(* IEC 61131-3 sources: ml2plc/benchmarks/st (part 9) *)

(* ---- LSTM2.st ---- *)
FUNCTION_BLOCK LSTM2_FB

    (* Model Inputs/Outputs *)
VAR_INPUT
    input_data : REAL;
END_VAR

VAR_OUTPUT
    output_data : ARRAY[0..2] OF REAL;
END_VAR

VAR CONSTANT
    weights_0_i : ARRAY[0..31] OF REAL := [1.39262271, 2.07329702, 2.0091362, 1.70178938, 2.3850913, 1.12900257, 1.77114773, 1.79174864, 1.94517601, 1.90923738, 1.87943172, 2.05496025, 2.01677155, 1.98114431, 1.29512143, 1.9032824, 2.06803155, 2.26776886, 2.24906993, 2.35914302, 2.58031249, 0.854317784, 2.0349102, 1.86201072, 1.96425331, 1.27948534, 2.47761846, 1.86080444, 2.06046557, 1.88541865, 1.78743565, 2.44109106];
    recurrent_0_i : ARRAY[0..1023] OF REAL := [-0.134004354, -0.148313314, -0.0194474477, 0.0388797, -0.0824599266, 0.0315496214, -0.173172131, 0.0359949544, -0.200757176, 0.109297805, 0.0659822822, 0.0169876534, 0.254330784, -0.00428949948, 0.129118174, -0.0437734537, -0.0245252717, -0.0815731362, -0.0834033787, -0.077183038, -0.0660836324, 0.0495678931, -0.029196145, 0.03283979, 0.0261739939, 0.0130877821, 0.106014706, -0.057191126, 0.0592699833, 0.0329136439, 0.216046751, -0.0511060841, 0.0071357484, -0.0244121794, 0.0280594658, -0.0301723629, 0.0475499704, 0.0748397335, -0.0587395504, -0.168087989, 0.161314234, -0.0552050099, 0.0945079327, -0.107845977, -0.0959540233, 0.00252881669, 0.139446095, 0.0318621695, -0.111325473, -0.0973692015, 0.0295887217, 0.000735154259, -0.0220976807, 0.0224685688, -0.0352836587, -0.031947881, 0.0713648722, -0.147181049, -0.041276142, 0.163752452, 0.163126245, -0.0694158077, -0.0533319078, -0.0770015121, -0.170238152, -0.178571403, 0.0332847945, -0.0801878721, -0.0456461273, 0.0202053282, -0.0822198018, -0.117651939, -0.0558106229, 0.0733473897, 0.0299465898, 0.0360525213, -0.0536533296, 0.0635128692, -0.0457392968, 0.126843438, -0.0655647293, 0.0488459691, -0.0775968879, -0.170379788, 0.061554566, -0.137451679, -0.115184806, -0.00126610929, 0.0082264822, 0.0221565478, 0.049042806, -0.0857262686, -0.0540655181, -0.090015851, -0.238347262, 0.050842043, -0.170883492, 0.0547744632, 0.042925328, 0.066795744, -0.090761885, 0.0645720959, 0.0878244713, 0.195313513, 0.00631635636, 0.0690589845, 0.131412268, -0.0195933655, -0.00472750515, -0.00867333263, -0.0322425812, -0.0256382748, -0.137210175, -0.00508641265, 0.0411479399, -0.0136672538, -0.188457325, 0.110275678, -0.0535120554, 0.148506701, -0.0941733867, -0.0840847343, -0.203250527, -0.00964725297, -0.0456403047, -0.0917202309, 0.0857251734, -0.142379165, 0.0902288333, -0.0697477087, -0.25946781, 0.200249165, 0.0577523112, 0.0731128231, 0.149998024, -0.0543648489, 0.160912603, -0.040147312, 0.0467842557, -0.00688959006, -0.0149163418, -0.0740291998, -0.0424987338, -0.0501250215, -0.076917544, -0.0832854882, 0.129720092, -0.00917770341, 0.154316008, -0.0984195694, 0.0695591345, 0.0279394947, 0.117725901, 0.0648251921, 0.120997198, 0.00961737428, -0.0130183501, -0.0333279334, 0.049932152, 0.0741841197, -0.0766564682, 0.0841158479, -0.0490418077, -0.00928253029, -0.0196176413, 0.131710216, -0.178811699, -0.0807049945, 0.0945211127, 0.0813005269, 0.0478863083, -0.0749040321, -0.0155161619, 0.0436361209, -0.0399981439, -0.00584720029, 0.219137162, -0.0570646003, 0.0864072666, 0.0547209121, 0.19448778, 0.11035566, -0.0152758295, -0.151405767, 0.0672118068, 0.0867983252, 0.0845759436, 0.0431055985, 0.0178876277, -0.055806689, -0.0743876174, -0.0819625705, -0.0752747655, 0.0704117194, -0.00382922404, -0.0398440622, 0.0417721309, -0.0862388536, 0.0705794618, 0.0484335832, 0.173169613, -0.00238036085, -0.0258361753, 0.148217037, -0.0232884251, 0.0270024538, 0.0563735589, 0.126127064, -0.116592243, -0.054894805, -0.174138799, 0.095002085, 0.0277814362, -0.046509631, 0.00551629113, -0.0126956999, -0.034402471, 0.11015445, 0.0495837145, -0.161556005, -0.0879831612, -0.0552681759, 0.0285979733, 0.163931042, -0.0467763692, 0.101849534, 0.0563726798, -0.0478363261, -0.0134126432, 0.0839114934, -0.185348555, -0.0519256219, 0.0111938342, -0.0469942242, 0.0292907096, -0.0607635677, -0.0199214034, -0.0835910067, 0.0188902467, -0.0856332853, -0.0664014295, -0.150778636, 0.232508123, 0.0984602422, -0.112400122, -0.0707815066, 0.00367648201, 0.0512798317, -0.109921589, 0.207549274, 0.162023827, -0.0390811004, 0.0424390286, -0.0276059639, -0.0962381288, 0.0657916293, 0.122452855, -0.145714879, 0.156922311, 0.174932122, 0.104362868, 0.0848342478, 0.0143698901, 0.0799010321, 0.106308773, -0.235139385, -0.082570672, -0.20124191, -0.0119339572, -0.0909275711, -0.0578141734, -0.10269203, -0.093932122, 0.0914303064, -0.107989773, 0.187612101, -0.01330359, -0.0776220039, 0.0276991762, 0.151062503, -0.0498313829, -0.067400828, -0.00874477439, 0.0098327212, 0.0279471185, -0.134616643, 0.102443077, 0.00515093608, 0.0774946585, -0.0788893849, 0.0691870078, 0.0495144166, 0.0123116644, 0.134680301, 0.0235169455, 0.0158374831, -0.0700131357, -0.0892158076, -0.00706590153, 0.00756208412, -0.0815098733, 0.16224964, -0.0743651763, -0.147885278, -0.0525642671, 0.0721946955, -0.00837692246, -0.077373594, 0.0789944157, 0.0923940986, 0.161076784, 0.0733315349, 0.100722194, 0.0398540571, -0.0822396129, -0.113960207, 0.117588356, 0.0800742581, -0.0111245122, 0.0219515339, -0.0255101845, -0.124131009, -0.240380466, 0.0300145727, -0.2196614, 0.0195070971, -0.0691136047, -0.0881249011, 0.0897721574, -0.125163659, -0.190538183, 0.00175063859, -0.0439649113, 0.119778425, 0.0073960349, -0.0287520792, -0.0209456533, 0.00432721013, 0.195701689, -0.0492347032, -0.0886455923, -0.0122433417, 0.0998576805, 0.0985153913, -0.0163457133, -0.0628783479, -0.195168257, -0.0639438778, 0.164951876, -0.112278, -0.0480273664, 0.0445793085, 0.0903970227, -0.137500077, -0.0213923361, -0.0938236639, 0.0234163329, -0.0859521851, 0.0565886721, -0.1431977, 0.0418196842, -0.0795657262, 0.118214853, 0.00396145741, -0.139788032, 0.133322746, -0.025860507, 0.0901994631, -0.132371172, -0.0476551503, 0.0196201466, 0.0488258637, 0.048791565, 0.0862637311, -0.0668302327, -0.0286542438, 0.0713004172, -0.0974688083, 0.0134516265, 0.10718289, -0.0149930362, 0.0711589083, 0.047025796, 0.035104014, -0.055901099, 0.0565550551, 0.148158491, -0.123526365, -0.228604481, -0.161055535, 0.133236721, 0.180309668, 0.0573264062, 0.024110429, -0.0977662504, -0.0378237776, 0.161678582, -0.0324702784, -0.0193747114, -0.0399733596, -0.0443898179, 0.136378944, -0.0683534667, 0.037007682, 0.204772562, 0.0150840413, 0.00119091454, -0.115353808, -0.0508661531, 0.0945357457, 0.00397635065, -0.0107160192, 0.0445148945, -0.153324053, 0.0779764131, -0.0182528608, -0.134156778, 0.113704324, -0.042016793, 0.0408653244, -0.0345638283, -0.104644932, -0.00025787577, 0.195931494, 0.0634211004, -0.0954237133, 0.000879314728, -0.119162239, 0.0455557369, -0.181164652, -0.0286782533, 0.0838612989, 0.00807927363, -0.149410591, 0.0170738958, 0.00178633351, 0.0720130056, 0.0684362873, 0.104216136, -0.0513023771, 0.011758212, -0.176010668, 0.0966927707, 0.0102190599, -0.0279936772, 0.043596521, -0.0417424887, 0.128085271, -0.0604554452, 0.0849098563, 0.0585800111, -0.242956415, -0.163328066, -0.130404904, -0.121299736, -0.0171396304, -0.0231877025, -0.159575537, 0.0178560223, -0.0958106816, 0.0408961512, 0.144970998, -0.120266221, -0.0517051853, -0.0798958912, 0.0248777233, -0.0202759672, -0.00199979614, -0.149970502, 0.0858172476, -0.0259563103, -0.0816580132, 0.10286995, -0.056762252, 0.100706398, -0.0494532436, -0.0494545288, 0.0237438828, 0.0785808489, 0.103829391, -0.0987794846, 0.00639404636, -0.0520768799, 0.0490948707, 0.0426566862, 0.0361592136, 0.0612452999, 0.0584818758, 0.17560859, 0.0293737985, -0.049783133, -0.107105657, 0.108317658, 0.0812257454, 0.0484825969, 0.111484915, 0.0553024188, 0.00590429641, 0.0106472084, -0.0448202752, 0.0259227678, -0.0365177095, -0.0368360095, 0.0979937613, -0.0990265682, 0.0768370628, -0.00803940371, 0.0511335284, -0.10439276, -0.0556471385, -0.111525387, -0.0822637379, -0.158447728, 0.00631242804, -0.0898952037, -0.0103400107, -0.126665518, -0.12826854, 0.164742142, 0.126374289, -0.0623154193, 0.105801776, -0.0670462921, -0.0859524906, -0.165727615, -0.108836487, -0.0711561739, -0.181308746, 0.0773165002, 0.0591216311, 0.0504512489, 0.00781396218, 0.0489371642, 0.112477235, 0.15160735, -0.012935142, 0.131209746, -0.117033251, 0.0818329602, -0.00354715297, 0.10224212, 0.107696757, 0.00897218473, -0.0807351544, -0.00682571437, 0.0395227484, -0.0326741263, 0.00277444068, 0.074753195, -0.0773364604, 0.100228824, -0.0078582773, 0.0254640095, 0.139588684, -0.136924639, 0.0528058484, 0.0296735466, -0.0419536792, -0.0416563302, 0.0534628034, -0.0191842429, -0.0148097789, 0.0523376055, -0.0542180687, 0.0964108631, -0.120417021, 0.038016621, 0.171443269, 0.100414015, -0.152942792, 0.13210088, 0.0675438419, -0.0117004402, -0.0681549385, 0.140697092, -0.0568291806, -0.0730812475, -0.118596427, -0.0816021189, 0.00568043999, -0.0364705734, -0.0795824528, -0.268455297, -0.00127396476, 0.185255677, 0.0253919102, 0.0383441038, -0.0536498129, 0.0324265659, 0.130935684, -0.0526439697, 0.0885849223, 0.0233933069, 0.111991353, -0.0564337634, 0.0322036669, -0.0236973744, 0.138340235, 0.0345056728, 0.0483544394, -0.0399727114, 0.0238587521, -0.0200702958, -0.0636315271, -0.178390726, 0.093400903, 0.0741568655, 0.0728121176, 0.0038592096, 0.0566493496, 0.191387981, -0.0285235178, -0.0280888584, 0.0401902087, -0.0860493332, -0.0164414719, -0.077161938, 0.00620657578, -0.0703452677, 0.0302030519, -0.038376864, -0.0379175022, -0.129299313, 0.0864133611, 0.112249866, 0.00572548434, 0.14621374, 0.0301852543, 0.149874419, -0.0408704281, 0.162906498, -0.00662965514, 0.0628379807, 0.0268993415, -0.000689674052, 0.134167075, -0.313462943, -0.0514584668, -0.107852802, -0.00314436248, 0.0118370224, 0.0500866398, -0.092870526, 0.141352415, 0.0112507679, -0.00922824256, -0.0692459121, -0.00235652924, -0.0174207557, 0.154500976, 0.081347324, -0.00308398576, -0.00189885148, -0.0499526374, -0.0560274385, -0.0403530262, -0.15555121, 0.0442879125, -0.059743192, 0.00816269685, 0.120614648, -0.00293097575, -0.0731150135, -0.0886584222, 0.0900309607, -0.115198389, 0.191818729, 0.103595406, 0.0381124802, -0.0148502458, 0.0115758171, 0.0609838217, -0.0460009836, -0.0733279809, 0.00619584089, 0.0253677219, -0.0612828694, -0.0889660418, -0.036679469, -0.155304044, -0.0361508727, 0.0593941361, -0.0159850381, -0.107755415, 0.205634415, 0.00516803795, -0.0302425101, -0.071119532, -0.0732871741, -0.00382628315, -0.0291780587, -0.0412666611, 0.0520398542, 0.000519843074, 0.177570358, 0.149022236, 0.10058704, -0.0362605043, 0.127544448, 0.0389988348, -0.0245497897, -0.0136824315, 0.0706591606, -0.0728941038, 0.0614774711, 0.0119364653, -0.133704841, -0.000918392092, -0.134823799, 0.0438350029, -0.00247984286, -0.0626151115, 0.09301278, -0.0666331053, -0.0263147596, 0.0359722786, 0.0305371247, 0.054677207, 0.0119109284, -0.0147482157, 0.00910742208, -0.129100755, 0.033809796, 0.00991856307, 0.00350326137, -0.10226763, -0.0163466893, -0.129900768, -0.135179013, -0.064366892, -0.0374643244, -0.0170351807, -0.0269057527, -0.0223082807, 0.0195573866, -0.154327378, 0.0836651251, 0.101992503, -0.266588628, -0.0957774445, 0.127723008, -0.0702769905, 0.000776129775, -0.0205887109, -0.0611850992, 0.102223888, 0.0193744767, 0.0702703893, -0.0131372688, 0.0499369912, -0.13509807, -0.00585971214, -0.0526572391, -0.0965908021, 0.122484364, 0.0293788202, 0.0450509749, -0.0484344773, -0.0140484432, 0.154743597, -0.0609884039, -0.132091016, 0.0942119583, 0.106592871, -0.12995939, 0.0108766314, -0.0612348542, 0.14751406, -0.112796851, -0.0632852614, 0.10222663, 0.00354706054, -0.033328332, -0.124713257, 0.0113556404, -0.279741585, -0.0857560784, -0.157485113, -0.00395657308, 0.0653496161, 0.0413245782, -0.00413726456, 0.0122570768, 0.166194528, 0.111745253, 0.0223836936, 0.00864755362, 0.0349040143, -0.0376916379, -0.0457340293, 0.0522189811, 0.114521392, -0.0617210828, 0.0331743099, 0.115298331, 0.0447754115, 0.142697737, 0.0433601551, 0.0632954091, 0.0451230034, -0.269107699, 0.000234287232, -0.0699387565, -0.016104091, 0.080592148, 0.0290849321, -0.0106361397, 0.00810046121, -0.174048468, -0.085996531, 0.0171728451, -0.03814153, -0.0919195488, -0.0125079993, 0.00758307241, -0.0626493841, -0.00948416442, 0.113764353, 0.0411069244, 0.111225121, -0.00789413322, -0.0439041629, -0.054905504, -0.135183468, -0.0833396018, -0.0639307648, 0.00211562216, -0.0953369364, -0.163012341, -0.134885401, 0.081080623, -0.112399474, 0.0664561316, 0.0931484252, 0.0478505529, -0.0171904434, -0.0378614031, -0.0456895977, 0.12899968, -0.0597828738, 0.0834410861, 0.0139350276, -0.0282864664, -0.0769604295, -0.181071818, 0.214174002, -0.100946948, -0.0732517987, 0.0612714738, -0.197533071, -0.0227342471, 0.0388891399, -0.100754239, -0.00672170753, -0.0207819417, -0.110634871, 0.022637371, -0.01396285, -0.011750361, 0.00330980448, -0.0859773457, -0.000174265006, 0.129387438, -0.139958769, -0.156467378, -0.0922901556, -0.0325083025, -0.0625371039, -0.0629708767, 0.0614186861, 0.0192336366, -0.0547801182, 0.0301011354, -0.0588637106, 0.0513670668, -0.164495796, -0.00147821754, -0.0780117661, 0.0552018546, 0.109413944, -0.00130969961, -0.00898661651, 0.0132659879, 0.0631986111, 0.0843208879, 0.061540179, 0.0394076332, 0.0400769822, 0.00576977246, -0.0982378572, 0.0421557277, 0.113608956, 0.0188576393, -0.0243477058, 0.0602114797, -0.0545240231, -0.0897894204, 0.101281449, -0.154307395, 0.135896564, 0.0464510098, 0.00640968326, -0.021830542, -0.0177672878, -0.0721066073, -0.309531212, 0.0388812348, 0.145754725, -0.0283625945, 0.0946166068, -0.154452384, -0.0263472404, 0.0116467727, -0.0632445514, -0.0424361527, -0.0449868031, -0.0440483689, 0.162283525, -0.141732365, 0.0662780777, -0.0210850425, -0.0168101434, 0.214176998, 0.15372856, -0.0118867746, -0.062056452, -0.000693539158, 0.104848668, 0.120308466, 0.0414873511, -0.112575084, -0.0714760497, -0.0417096615, 0.222792968, -0.110523865, 0.0548756756, -0.117230386, 0.0457057953, 0.0473512486, -0.0799265727, 0.105714075, 0.0468949117, -0.132061332, -0.0291638914, 0.102133185, 0.0477667376, 0.0171793289, -0.0337885171, 0.151557818, -0.0374314077, 0.0159622598, 0.194910049, -0.0489041544, -0.133889884, -0.11275547, -0.173466712, -0.0138423145, 0.13869071, 0.0596037172, 0.062202137, -0.0821835101, 0.0251389612, 0.0879076049, -0.0829390064, 0.0959333256, -0.0619588941, -0.141935766, 0.114354968, 0.155747041, 0.00375959137, -0.0630423576, 0.0245623328, -0.0128721073, -0.103164501, -0.000736813992, 0.0574771278, 0.083872661, 0.0506197587, -0.0941908583, -0.0433398113, -0.00233667111, -0.0455719605, 0.0782523602, 0.173237547, 0.0224949233, -0.0517513119, -0.0378127173, -0.0389218852, -0.0414382815, -0.166335255, -0.110787965, -0.0431358181, 0.0556307398, -0.0059117917, 0.00672180811, -0.00877491664, 0.0884027109, 0.0815280005, 0.0644761026, -0.0395023786, 0.145024762, -0.152458549, 0.0229760204, -0.0113443667, 0.178633645, 0.0435204618, -0.119631179, -0.155641362, 0.169697255, -0.0196635164, -0.0875597149, 0.0888158455, -0.0858875215, 0.112062834, -0.0394157432, -0.120597802, -0.0225557201, 0.0881219059, 0.0495140031, 0.0828080699, 0.00243129907, 0.0277386475, -0.00106827542, 0.0104990676];
    bias_0_i : ARRAY[0..31] OF REAL := [2.26711226, 2.27420187, 2.30581617, 2.31258035, 2.41937995, 2.14668489, 2.35069036, 2.0788188, 1.95626056, 1.9590205, 2.35707855, 2.41049099, 1.97553778, 2.61581278, 2.24078465, 2.34379292, 2.58412099, 2.61249423, 2.82780743, 2.28536749, 2.70651102, 2.23035336, 2.46460962, 2.46926284, 2.27272534, 2.30647492, 2.72902465, 2.39153671, 2.38868213, 2.66885066, 2.01619935, 2.59971189];
    weights_0_f : ARRAY[0..31] OF REAL := [-0.103510261, 0.155920088, 0.000336945057, 0.0438489616, 0.0438292921, 0.0684255958, -0.0156891793, -0.0915879682, -0.150318235, -0.0157852769, 0.165699959, -0.0541729182, -0.130850449, -0.102231637, -0.09064731, 0.185210466, 0.0596044362, 0.0255541503, -0.132748216, 0.168993115, 0.0778170228, -0.178415745, -0.0980168432, -0.111201935, 0.00410218537, 0.0909076929, -0.19583635, 0.177583277, -0.195816249, 0.05490008, 0.129835844, 0.0483838022];
    recurrent_0_f : ARRAY[0..1023] OF REAL := [-0.00691014668, 0.0539467856, 0.0330422595, -0.0597359128, 0.0169141795, -0.0331418402, 0.0173334759, -0.115839541, 0.0169229154, 0.00140885415, 0.0407177694, -0.0358268954, -0.109294459, -0.144246504, -0.000686382409, -0.112673983, 0.204203159, 0.151690304, -0.0307787433, -0.0266794655, 0.118159838, 0.0687537044, -0.196012646, 0.125656754, -0.0728332177, -0.110024385, -0.0255501121, 0.0337689295, 0.12247669, -0.00833526812, 0.0699421838, 0.10112042, -0.0160470735, -0.251208723, 0.0141219553, -0.104823828, 0.0795288607, 0.146455094, 0.193343654, 0.0469122157, 0.00523563568, -0.0152252698, 0.107677527, 0.0577447973, 0.203866184, 0.0566105619, -0.0699815378, 0.0103690829, -0.025823988, 0.0698903576, 0.0937844068, -0.0525806397, -0.0100893909, -0.00210557133, -0.027120579, -0.125489399, -0.0150436275, -0.137994111, -0.0517354123, -0.00446202187, 0.0964010805, 0.0635783747, -0.179122448, -0.0195943583, -0.0458602905, -0.117201932, -0.104822852, -0.0428061485, 0.102384202, -0.0332811326, -0.0195743572, 0.139496908, -0.227235973, -0.0425146483, -0.0722654611, -0.00887431018, -0.132653967, 0.0553128608, 0.112583086, 0.165537104, 0.0365887061, -0.101447128, -0.0985822976, 0.134091511, 0.126952991, -0.0307374429, 0.156312183, 0.0430723652, -0.0509468019, -0.0238420386, 0.0764375478, -0.156924069, 0.207784161, -0.0545833334, 0.0418132134, -0.0283788238, -0.0884652212, 0.0490699746, -0.0942642987, 0.0732667968, -0.030637661, 0.070327282, -0.0578977019, -0.00136273983, -0.0913911015, -0.0634720176, -0.00320455851, 0.0674236417, 0.153130755, 0.0737068728, -0.058094427, -0.0211398825, 0.047294125, -0.0165242814, 0.0421787389, -0.194994301, -0.00844584592, 0.224502295, 0.0124900211, -0.0566204153, 0.14547962, 0.0214617066, -0.0670055449, 0.0452741906, -0.0959712192, -0.20302707, -0.12255279, -0.121577464, -0.243490487, 0.111299828, -0.0271219537, -0.138370499, -0.00303730182, 0.0865178406, 0.036418654, 0.0138794044, 0.168218017, -0.0838619396, -0.0444532298, 0.0891045108, 0.00708426163, 0.0661141723, -0.0399264023, -0.196934208, -0.00761342235, 0.0918690488, -0.0572661683, -0.19526419, 0.0615054481, 0.0232604593, 0.0763470009, 0.00757205719, -0.170795515, -0.0579727553, -0.176360965, -0.0789391994, -0.100149475, -0.065748468, 0.155853912, 0.212572694, 0.0898325294, 0.0844217762, 0.0629207939, -0.0372571982, -0.0432355106, -0.181974009, -0.0866544694, 0.0077539701, 0.0990353674, 0.0708501711, -0.0190058965, 0.0995751917, 0.0896994844, -0.00912527274, -0.0338458568, -0.0137675917, 0.0123393871, -0.0475793704, 0.00175741455, -0.0418805219, 0.115797728, 0.102187678, -0.119467586, -0.0719964802, 0.0550041869, 0.0517715327, -0.0794643909, -0.0289103501, 0.162206873, 0.0127481343, -0.158131227, 0.0304524321, -0.0849102885, 0.0366410948, 0.00384486257, 0.00391263934, 0.0273174196, 0.0815227702, 0.121064574, -0.0600702949, 0.0945892483, 0.057374645, 0.0601622164, -0.0795332193, -0.117707953, 0.0210899487, -0.0372100323, 0.0654684305, 0.0984267443, -0.105141684, 0.138595685, -0.242979154, 0.0243996978, -0.146832377, -0.0938290209, 0.0239801873, 0.124723487, 0.0749439299, 0.0199104045, -0.0626129135, 0.0605645701, -0.112765379, 0.183117643, 0.0728753209, -0.0168619975, -0.0250719804, 0.055014126, -0.0111222807, -0.0467175767, -0.120118842, -0.0719998553, 0.0297824219, 0.0637432635, 0.0930763558, 0.13979651, -0.0786714107, -0.0663307607, 0.0274352431, -0.0654640198, 0.0392157845, -0.0611319244, 0.0636766329, 0.0744584575, 0.0101938117, 0.0555800907, 0.0684161484, -0.0313910916, -0.0375169925, -0.0980222523, -0.138520613, 0.0849486813, -0.1236277, 0.229274869, -0.106394686, -0.104073107, 0.14711982, -0.108186357, -0.0884629786, 0.00385326333, -0.0557541102, 0.0872948691, 0.107587278, 0.0581731871, 0.0215235408, -0.0997304693, -0.0756542683, 0.111098066, 0.0226193108, -0.116672814, 0.0418509804, 0.115937918, -0.0735490248, -0.110052764, 0.063148357, 0.00697960611, 0.0338207707, 0.217933804, 0.059628129, -0.00196746015, 0.123881862, 0.117818907, -0.0192651134, -0.0493695848, -0.0318081304, -0.0192032102, 0.0678166598, -0.00145450607, -0.0869160444, 0.164906725, 0.0981748998, -0.0928812325, -0.0604305677, 0.104643285, -0.142461985, 0.0815763474, -0.00508458167, -0.115501776, 0.0773961246, 0.269783676, -0.172341615, 0.153024822, 0.0490144491, -0.0540101454, -0.0356579125, -0.0566640384, -0.0655708835, -0.0586362667, -0.188088432, -0.0623720735, 0.0904100835, 0.0650910586, -0.0290365405, -0.05520254, 0.0847302079, -0.0487206914, -0.0588986054, 0.0449058786, -0.0469482914, 0.00918797776, 0.0142356111, 0.0266836565, -0.138558552, -0.0684637055, -0.106428206, 0.0228035878, 0.00893711299, 0.00322866905, 0.0695354939, 0.0546293296, -0.0871017501, -0.0162100531, 0.0719157681, 0.0608419478, 0.0179101136, -0.111390203, -0.0720891654, -0.0755965486, 0.0167733729, 0.0292966813, -0.123163752, 0.00929058343, -0.235721245, -0.0745700151, 0.0623340309, -0.0371385068, -0.0765249506, 0.0989028439, -0.139854208, -0.0925003365, -0.0397025943, -0.115456559, -0.116422005, 0.032429643, 0.0281777196, -0.0239272695, -0.0328503177, -0.144181833, 0.0372066684, -0.0524021909, -0.0436877087, -0.144946769, 0.0973152816, -0.107339486, 0.100682661, 0.0554906614, 0.0365729779, -0.0905715972, 0.098124668, -0.0407010354, 0.231915027, -0.103092752, 0.0268508829, -0.00293016527, 0.082363911, 0.0652320087, -0.0384592302, 0.12898241, 0.0402026586, 0.0469526425, -0.0367732197, -0.0941489637, -0.21039243, -0.0243418086, 0.0567742139, -0.0757714957, -0.224011689, 0.111577362, -0.0840680152, 0.00466096681, -0.0797860324, 0.0477439202, 0.0298575554, 0.0669026896, -0.0090283975, 0.112681448, -0.0502874851, -0.00540959276, -0.0274625272, 0.0441634879, -0.0369217657, -0.0101684844, 0.0535784513, -0.00723357126, -0.00442850217, 0.0174251013, 0.0924004242, -0.0299789757, -0.152222574, -0.142336786, -0.0262773167, -0.0686421767, 0.167089716, -0.0872355402, -0.0557465181, -0.113622896, 0.14195551, -0.0551547408, -0.0710106269, -0.067609705, 0.0912378356, 0.0599844456, -0.0631347969, -0.0533212051, 0.0721441358, 0.145896912, -0.0850262195, -0.0618097708, 0.029887341, 0.0855583772, -0.000903251348, 0.0312168524, -0.144762039, -0.0528443567, -0.0244600698, -0.138042107, -0.059540391, 0.0647165254, 0.116018802, -0.158837333, 0.0567534491, 0.0310964324, 0.0519501194, 0.166376859, 0.000156691065, 0.0405331813, -0.0376353115, 0.0910912305, 0.0336197764, 0.0320295431, -0.0283036716, -0.00967699476, -0.0228656419, -0.0633295774, -0.0474807657, -0.0476354286, -0.0262157004, -0.00842537172, -0.0226355828, -0.036474023, -0.144134447, -0.0138616599, 0.0502098948, -0.141214415, 0.0914947763, -0.211922467, 0.108886033, 0.0302329641, -0.0443936884, -0.024401769, 0.178851143, -0.0395925194, 0.109363601, 0.017790867, -0.0280343331, -0.00382982777, 0.00198424468, 0.0132888649, 0.0585306659, 0.0230387188, 0.0412786007, 0.0889222324, -0.122444734, -0.0592958406, 0.061345689, -0.0724695697, -0.17240414, -0.0215452053, -0.11073748, -0.161671206, 0.0069130389, -0.0864949152, -0.0884157494, -0.107923985, -0.149227038, 0.103861548, -0.0224465597, 0.024422098, 0.0677691996, -0.145919502, -0.0570074134, 0.0319532827, 0.0987191796, 0.0601408072, 0.0278520733, -0.146264344, -0.0350774638, 0.0202368796, -0.0724366754, -0.0483524352, -0.156716764, -0.0751653537, 0.0405076034, 0.106280632, -0.090791665, -0.0230285358, -0.0929582193, -0.111961611, 0.016109759, -0.0204031523, 0.0609163716, 0.136724174, 0.0567737892, 0.00902334042, 0.16077508, -0.124572918, 0.0124027627, -0.103831545, -0.0465113223, -0.057945013, -0.117938057, 0.0314415023, 0.0152452486, -0.0766829997, 0.0884116963, 0.0839675665, 0.0765219554, 0.0703505203, 0.0279270336, -0.0127789946, -0.0291803852, 0.0105592217, 0.0371113271, 0.0967723876, 0.0892940015, 0.103656046, -0.260149986, -0.0384903848, -0.0810357556, 0.0938086882, -0.0499689803, -0.0526683852, 0.0961615741, -0.00260981917, 0.00965978112, 0.0354677886, -0.0273469277, -0.0378791988, -0.0684229508, -0.153382406, 0.0829801634, 0.0420659184, -0.0491692908, 0.0548881516, 0.0939008445, 0.0785935223, 0.072916232, -0.0753023624, 0.101734571, -0.212460309, 0.216674268, -0.0828238726, 0.179046914, -0.0126461163, -0.0996344835, 0.0554261804, 0.0543882214, 0.0894713178, 0.0131856054, 0.18864961, 0.0088903252, 0.133240402, 0.0488812737, -0.0503490269, 0.120177239, -0.12674436, 0.0911346078, -0.204793841, -0.0583979376, 0.0430473685, 0.0117439311, -0.100650795, 0.0597399846, -0.183556691, 0.0328893699, 0.0997276679, -0.162350491, -0.0379387476, -0.0467698462, 0.057570409, -0.0352495015, -0.0132564018, 0.0427324548, 0.0986689329, 0.0538132042, 0.000333502423, 0.0106591079, -0.106351398, 0.0680583045, 0.093219772, 0.028425552, -0.0404609889, -0.20924823, -0.127012178, 0.0357946232, -0.0195649005, 0.0538770743, 0.0498228967, -0.056039989, 0.0299009793, 0.0457624719, 0.0841314942, 0.00167563639, -0.0151560055, -0.0918175727, -0.0157458112, -0.252087355, -0.0610392466, 0.118945099, -0.0761914626, -0.059865877, 0.0874174461, 0.145287514, 0.0177363213, -0.207373992, -0.158034712, 0.0130132614, -0.0213055164, -0.110472739, -0.0698485523, -0.00191319175, 0.026409829, -0.149118632, 0.0352956653, -0.0690959916, 0.0712720454, 0.0497274585, -0.0684742928, -0.0192867741, 0.0131304041, 0.0943724513, -0.158797354, 0.0100931283, 0.0212941729, -0.173423976, -0.0672471523, 0.0538061112, 0.125850394, -0.0581939593, -0.0356761925, 0.101517476, 0.0305221472, 0.072131291, -0.051977843, 0.0737764239, 0.0950229913, -0.0675911531, -0.098661676, -0.134873658, 0.0323955193, 0.093537353, -0.0435548872, 0.0345223173, 0.0441020727, 0.0258881748, -0.0267370548, 0.0141971605, 0.0358532406, -0.124594763, 0.0248470921, -0.0100919018, 0.0500047579, -0.0708093271, 0.128508076, -0.0366209187, 0.106708124, -0.00206466648, 0.0805527717, -0.122561544, -0.0874712169, -0.0383777618, -0.0786395073, -0.0780212358, 0.0687881485, -0.0462901331, -0.0869080275, -0.0328290574, 0.114670701, 0.1203302, -0.0302833952, -0.0977141485, 0.0308538172, -0.054454051, -0.0955775306, -0.0812499896, -0.0532917529, -0.047714889, 0.0148271862, 0.0594015457, -0.0969915688, -0.0696531162, 0.0647605136, 0.0158956926, 0.00915151369, 0.16740869, 0.111624435, -0.0313705765, -0.126204967, 0.166225314, -0.00429002754, 0.00159279886, 0.170427188, -0.0651404411, 0.0322218463, -0.107634276, 0.110197365, 0.0253799651, 0.0844260231, 0.109976798, -0.0586437285, 0.0578876138, 0.000859050546, 0.189837858, -0.0570421889, -0.170068368, -0.0814624578, -0.0846147761, 0.0692067817, 0.0624997802, -0.227033526, -0.0656075999, -0.0454960801, -0.0364593938, -0.0984016657, 0.139481351, -0.0299721137, 0.0211200267, 0.0929757655, -0.162706748, -0.192191154, 0.194119602, 0.146404952, 0.0726765618, -0.0705825686, 0.000404240564, 0.00767246261, 0.0835697502, -0.0302281529, -0.0174284484, 0.0485032201, -0.120143197, -0.108964629, 0.0507510044, 0.00870033167, 0.0645659417, 0.108325213, -0.0504615642, -0.0399887264, 0.0522538908, 0.103842363, -0.0575898327, -0.0733171329, 0.0778556466, -0.0311737508, 0.000791670987, 0.053147953, 0.000775715336, -0.0727582201, 0.059283942, 0.015961254, 0.0980835333, 0.153303385, 0.0523465499, 0.200393319, -0.0961034298, 0.00924751814, -0.102561079, -0.127784446, 0.0216288883, -0.0499887094, 0.0408567637, 0.0934649706, -0.0518678166, 0.132874012, 0.0137811955, -0.05145818, 0.0129512828, -0.139415756, -0.143087536, 0.068125844, 0.10787306, -0.057314042, -0.0380743705, -0.0627397448, 0.130972728, -0.0196755826, 0.0785539597, 0.122383311, 0.0626117215, -0.0613358766, 0.0130844237, -0.0416473523, 0.0771606714, -0.053707961, 0.0782196, -0.00344187161, 0.102742925, 0.0139414081, -0.155407608, -0.0412477255, 0.0853889138, 0.063173607, 0.116590202, -0.110537179, 0.00120887649, 0.112075336, -0.0691253319, -0.0917270258, 0.0188949592, 0.00672117434, 0.0868049711, -0.121678926, 0.116180249, -0.0147003271, -0.0895797387, -0.135892138, -0.141551331, -0.212871507, -0.0520402603, 0.0142919831, -0.088278383, 0.0244035851, 0.0466132648, -0.0750784948, 0.106897034, 0.106365465, -0.0986929387, 0.168738917, 0.0507040955, 0.00279272767, 0.0927622467, 0.226838261, 0.0705733225, -0.152726993, -0.0682013631, -0.069567509, -0.106382623, -0.0238234401, 0.0889748037, -0.095707342, 0.0320834182, 0.0533372127, 0.0397444218, 0.173014328, 0.114501618, 0.050176464, 0.0578774475, 0.0132526672, 0.100262016, 0.113684908, -0.127054498, 0.016781047, 0.105807446, 0.160546854, -0.0204436425, 0.0449761264, -0.00650018919, -0.0162856318, -0.031046655, -0.00719706295, 0.17228359, 0.0929863527, 0.112568557, -0.0106027573, -0.0801606029, -0.00430984143, 0.0905482695, 0.102497414, 0.022951575, -0.0023685242, 0.101059511, -0.123741455, -0.0253990814, 0.00617785938, 0.224820018, 0.0564163029, 0.0227698721, 0.0183891784, -0.193179756, -0.048081845, -0.00418907218, -0.0182756223, 0.0594953559, 0.116223007, 0.083689943, 0.0758306682, 0.0600401387, 0.0057036127, -0.119169444, -0.00241687289, 0.049240943, 0.0222266763, 0.0222300421, 0.0184250548, 0.137113541, 0.133112341, -0.0405313745, 0.0703310296, -0.0368162692, -0.00698137842, -0.0782028064, 0.154308647, -0.0416583829, 0.0667509288, -0.0523070544, 0.000271657365, -0.148217291, -0.011399786, 0.0411178507, 0.0403273664, 0.182938606, 0.00969816186, -0.0497058183, -0.0412162356, -0.0586917587, 0.136667043, 0.0978190973, -0.0634948984, 0.0585792921, -0.0983795375, -0.0980659947, 0.0711884275, 0.0689789802, -0.109272763, 0.0259555485, 0.0922681913, 0.0452702269, 0.0214219354, 0.0569992065, 0.0292213559, -0.0258827768, -0.0412379466, 0.147309318, 0.0441662334, -0.0152443759, 0.00304972567, 0.182876348, 0.164139763, -0.111702725, -0.0858073086, 0.0243306477, -0.0263965055, -0.08150056, 0.0267791264, -0.0301363561, -0.110263094, 0.0477498025, 0.0285967328, 0.0422384776, 0.145023987, -0.0232882276, -0.109742552, 0.0407254286, -0.101167023, 0.087719284, -0.144451484, 0.0783894286, 0.116550274, -0.0671435595, -0.0849284753, -0.00986922067, 0.0360355005, 0.161055446, -0.118753619, -0.0674274117, 0.0250015743, -0.0504739732, 0.136040404, -0.160468519, 0.0275609754, -0.0788998529, -0.0405119434, -0.00997654907, -0.061767187, -0.053517133, -0.0994137824, -0.0556045212, -0.0925223976, 0.161830351, 0.0968106836, 0.0508179069, -0.0246349927, -0.0123783387, 0.0485562719, -0.0574627705, 0.0263824128, -0.120863646, -0.0710439906, 0.0614336506, -0.106016003, -0.0335879326, -0.0433921926, 0.0639650673, 0.0271945707, 0.0527300388, 0.0320915915, 0.013170423, -0.08443138, 0.248558924, -0.0503826216, 0.106785677, -0.046431087, 0.103803217, 0.0041458183, -0.0421562381];
    bias_0_f : ARRAY[0..31] OF REAL := [1, 1, 1, 1, 1, 1, 1, 1, 1, 1, 1, 1, 1, 1, 1, 1, 1, 1, 1, 1, 1, 1, 1, 1, 1, 1, 1, 1, 1, 1, 1, 1];
    weights_0_g : ARRAY[0..31] OF REAL := [1.47532678, -1.70458651, -1.47144258, -1.44691277, -1.68858755, -1.54678094, 1.4575063, 1.77509093, 1.5990113, 1.71160305, -1.5320437, -1.79037261, -1.77602446, 1.70425713, 1.4617672, 1.54794741, -1.52839839, 1.55297565, -1.90853524, 1.71287596, -2.10243273, 1.36646223, 1.82073891, 1.9412576, -1.69837666, -1.66724396, -1.99537337, 1.69469917, -1.80649602, -1.47025287, 1.49180543, -1.93371117];
    recurrent_0_g : ARRAY[0..1023] OF REAL := [-0.101195998, 0.08740969, -0.104587115, -0.16821076, 0.174443915, -0.035774447, -0.0947507322, 0.0378404111, 0.0557015277, -0.0394512936, -0.207284242, -0.197577581, -0.0711208954, -0.120538749, 0.0129681649, -0.0769899487, -0.0140917841, 0.00214586221, 0.00265539065, -0.123874903, -0.107705243, -0.105937153, -0.0518222116, -0.0369259045, 0.0763554201, -0.0299211461, -0.0788105503, 0.117140636, 0.00431261165, 0.0359783769, 0.00918749906, -0.104668915, 0.061548844, -0.0556093194, -0.0334143862, 0.0841006264, -0.0666153282, -0.0459342971, -0.0507918485, 0.0554375648, 0.0217144638, 0.0350073129, 0.124298088, 0.0216758177, 0.120086238, 0.0596877821, -0.0242632702, 0.0876686648, 0.0902777761, 0.0481038094, 0.204886943, 0.180912375, 0.0283590574, -0.00545403361, -0.111476384, -0.0184426904, 0.0296593215, -0.0534377694, -0.0470365658, -0.0600505061, 0.0377211198, -0.0949909091, 0.160191432, -0.0323576629, -0.00774259027, -0.000638007885, -0.0570991226, -0.00242817705, 0.0460335501, -0.0124942036, 0.255657285, 0.0184760075, 0.083474122, -0.138274193, 0.0288563892, 0.0561495312, 0.10814105, -0.0252166167, -0.083617121, 0.00315840216, 0.134269193, 0.080687955, 0.0888233185, 0.0208418351, 0.0151973907, -0.0696730837, 0.254600137, -0.126226783, 0.00475102197, 0.0205613524, 0.0766184479, 0.0583407693, -0.0356217064, 0.0329036042, 0.00880802702, 0.0259327479, 0.0302957594, -0.0485900454, -0.0475254133, 0.0427846983, 0.14055638, -0.125194758, -0.230593339, 0.115369402, -0.009178821, 0.0961865857, 0.0861247405, -0.0569514222, -0.0642841905, 0.0787181482, -0.000574963633, 0.00898596738, 0.0703639537, 0.0666252524, -0.082310304, 0.0077218432, 0.0239734557, -0.154473484, -0.130902037, -0.138917118, 0.168707773, 0.0168054793, -0.241201326, 0.0562871881, -0.0551889241, 0.0774001628, 0.0454477295, 0.0527046323, 0.192182556, 0.0634233505, 0.0726593807, -0.0730486736, -0.046287708, 0.0937241539, 0.155822381, -0.0986693949, 0.10592638, 0.0549062192, 0.0108801452, -0.0758548081, -0.150141403, 0.000112835725, 0.168501094, 0.0566198267, -0.000829054043, 0.081648834, 0.0720061287, 0.00562748406, -0.0315910913, 0.0916485265, -0.0881970823, -0.0454844274, 0.115997486, -0.0706517994, 0.200185716, -0.212817028, -0.266671538, 0.0280515496, -0.0507685766, -0.0832299516, -0.0272886436, -0.0584619641, 0.0404174477, 0.139308289, 0.104658842, -0.083959721, 0.0130339842, 0.0628424138, -0.0578840524, -0.0111292899, -0.0674168542, -0.0567888021, -0.0487619378, 0.0660481378, 0.140314907, -0.103330687, -0.077637881, 0.0232625715, 0.16300194, -0.0148641821, -0.121850781, -0.0120066088, -0.120630994, 0.0325469822, 0.00378151797, 0.0231334269, 0.0288972799, 0.117997028, -0.00443882123, -0.154459015, 0.0336177275, 0.0930437893, -0.00218074629, 0.131201416, 0.095992431, 0.115522057, -0.0244959947, -0.00682251481, 0.0696546957, -0.0206905808, -0.0148855159, -0.0281523354, -0.03817432, 0.0418252461, 0.0572236478, -0.0574149303, -0.109414637, 0.0453919359, -0.000927357178, 0.0428337641, 0.0247878674, 0.0959960148, -0.00927572511, -0.0164810531, -0.116284199, -0.0459703058, -0.0627707541, 0.0265134163, 0.0581545085, -0.00378958462, 0.0373996682, 0.0825420693, -0.0857948065, 0.0619786419, 0.081787698, 0.108454175, 0.0945709571, -0.051475592, 0.0921381786, 0.170338392, 0.137564644, -0.132172644, 0.0645276457, 0.154890299, -0.0760021806, 0.096898526, 0.0867238268, 0.109539069, -0.0057261046, 0.060632281, -0.100636743, 0.157683015, 0.0451725535, -0.00428324332, -0.0746827871, 0.0471339598, -0.0752350464, 0.069367975, 0.047093872, 0.00814475119, 0.011384381, 0.0659590662, 0.156899557, -0.0580012202, 0.085925512, -0.0214249622, 0.0120120468, 0.113536887, 0.0602683052, -0.0160956811, -0.0338802151, 0.0308419038, -0.0770991966, 0.000288646523, 0.0453838557, 0.0851812661, 0.0191567522, 0.0233700275, -0.121437192, -0.0659240335, -0.123420395, -0.0978944823, -0.0577415749, -0.0328979529, -0.0636603981, -0.00405571982, -0.0314529873, -0.020198442, -0.0146561153, -0.0762880072, -0.0999139771, 0.0514613762, 0.0256823711, -0.0942612588, -0.052791819, -0.133564845, 0.0861075073, 0.00868083257, -0.00935054384, 0.0302694831, -0.0317124836, 0.087807633, -0.0803157836, 0.089592196, -0.0941260234, 0.0717165917, 0.0632364899, -0.214625821, 0.137252107, 0.209107444, -0.117832825, -0.00798236765, 0.0595166907, 0.118651874, -0.108172223, 0.136428297, -0.18883127, -0.107870199, -0.0385832936, -0.206498623, 0.0613527596, -0.00105835567, 0.136841521, -0.0176947806, 0.00627136417, 0.0683735684, 0.0605167933, 0.0425770134, -0.00393029675, 0.00458816718, -0.0597686134, 0.0324797593, -0.0304794982, -0.0699171275, -0.0795711279, -0.0220978875, 0.11555858, -0.0186585672, 0.0740450099, 0.0289000161, -0.0231691636, 0.125412941, -0.0254150778, -0.0975785479, 0.0826669931, 0.0427691564, -0.0265431367, 0.0233916827, 0.0275735483, -0.159331188, -0.0835884213, 0.0867214575, 0.0581048802, 0.0400546007, -0.11298833, -0.0843894854, 0.0884476602, 0.156565502, 0.0398587845, 0.084373489, -0.167539656, 0.0533768237, 0.180099636, -0.0643721148, -0.022131959, 0.0352704972, 0.102284059, -0.129944429, 0.0652202368, 0.0329418108, 0.0671919212, 0.0213613939, -0.041750174, 0.140751526, -0.010692168, 0.108571574, -0.0590898506, -0.00340850884, -0.101751246, 0.0585011132, -0.0625699461, 0.0747210979, 0.143278256, 0.0285833869, 0.000918021193, 0.0832627043, 0.0124035478, 0.00828075409, -0.0645460263, -0.0208687484, -0.0479471907, -0.0879585519, 0.00869457796, -0.0489250496, 0.0110164564, 0.0660134107, -0.0409986079, -0.0835550651, 0.108670741, -0.0402804874, 0.0745845065, 0.0347721204, -0.0930110365, -0.0466776416, 0.0181542635, -0.122449115, 0.0457023606, 0.0551486239, 0.0993403047, 0.0452728644, -0.0912225768, 0.177634746, -0.0193397272, 0.0517804064, -0.078884609, 0.0770803168, -0.026274981, 0.115404844, -0.0222992562, -0.0548713244, 0.115336612, 0.102776915, -0.105107367, 0.0272116847, 0.0181901883, 0.116371438, 0.0772981793, -0.0657144263, 0.0702497438, -0.0933898166, 0.00560039189, -0.117238283, 0.043919649, -0.0706500262, -0.036055591, -0.103364304, 0.0620049611, 0.122532926, -0.0542505234, -0.0309813488, 0.112967849, 0.00626176875, -0.0412489027, 0.000259818044, 0.1122576, -0.022883717, 0.0698174983, 0.0954817906, -0.0475088432, 0.0141142579, -0.0512579754, -0.0754119679, -0.0424957797, 0.0419287719, -0.054218974, -0.156465426, 0.114787057, -0.0610668324, 0.0348946378, -0.040694993, 0.121415451, 0.0283232052, -0.0169020146, 0.139543638, -0.170662105, -0.119277015, 0.0594007708, -0.0582244582, -0.0817419291, -0.0981166661, 0.00173791777, 0.00693563698, -0.0207109731, -0.035633482, 0.0308553185, -0.0928787142, -0.0212399177, 0.0114278868, 0.136616603, -0.0549275205, 0.0995251387, -0.0262963269, 0.0154484715, -0.0506038368, 0.015139862, -0.0465807803, 0.0256181471, 0.0665449798, 0.0268637985, 0.136133835, 0.132263571, 0.0828409493, 0.00177018531, 0.188435555, -0.131212503, 0.0970125347, -0.127591342, 0.0796364471, -0.0402331352, 0.0689072907, -0.0653174818, 0.0493306741, -0.139246956, -0.0419746451, -0.0420375466, -0.133270577, -0.0126191825, 0.106959179, -0.0525025129, 0.0485690534, -0.0125091951, 0.0833685473, -0.0323823877, -0.0772480667, -0.0500528924, -0.204458624, 0.0348587632, 0.200497746, -0.0761522502, 0.0727544576, -0.0308812261, 0.0495476648, -0.146705776, 0.0997447371, 0.012238658, -0.00608632155, 0.150759101, -0.123230845, -0.0151646882, 0.0577027462, 0.0434368625, -0.0141762858, -0.200296491, 0.0534211285, -0.011844527, 0.189423949, -0.107985377, 0.0767114758, -0.135413483, -0.00799088273, 0.134802759, -0.0511588715, 0.0691743344, 0.105821721, -0.0770135447, 0.0278117098, 0.00748841185, 0.0431736782, 0.022644151, -0.0930894092, 0.0724659637, 0.119439431, 0.157009006, -0.110694274, 0.0888616964, 0.0203899164, 0.0554994904, -0.0155844046, 0.0935843065, -0.0437429696, 0.0356643498, -0.00294274278, -0.0150379483, -0.152130276, -0.0716923475, -0.221969858, 0.102691673, -0.0195766296, 0.0772279948, 0.0226173997, 0.0137649449, -0.0166043434, 0.116271779, 0.0191773064, 0.00167295639, 0.0734597445, 0.0365498513, 0.0512108281, 0.144751921, -0.0385083035, -0.0588598065, -0.189036906, -0.14177978, 0.0120348353, -0.0084497435, 0.220320597, 0.0226446763, -0.248947561, 0.139383212, -0.0020379154, 0.0696443245, -0.0780093148, -0.0792569518, -0.0160436984, 0.0795049742, 0.0932552516, 0.0753452033, 0.0848368406, -0.00240107533, -0.033641424, -0.0348135754, 0.0561227389, 0.147689387, -0.0594362281, -0.0409766734, -0.250746489, -0.160236001, 0.0386024341, -0.0686084852, -0.0440940112, 0.0674488544, -0.210844234, 0.0464956835, 0.0757730156, -0.0683382824, 0.0804399922, 0.0413802229, 0.0806305632, 0.0221607983, -0.132880241, 0.0989559144, -0.118918777, 0.0531449281, 0.0418806486, -0.0401233248, 0.0478454567, -0.0536536165, -0.00559705123, -0.0308934376, 0.0934929922, -0.0454997756, -0.121145718, -0.0170345623, -0.0106199561, 0.150425464, -0.0529386513, 0.067161046, -0.0163639486, -0.0500465147, 0.103452504, 0.0317030214, 0.0288870297, -0.011946328, 0.0184828602, 0.139818698, 0.101647899, 0.1074147, 0.0303774215, 0.134888709, -0.179935634, 0.036726281, -0.10821747, -0.142873049, -0.0262996051, 0.0476385057, -0.0365874916, 0.111659452, 0.0944161266, -0.0142952949, -0.0806843117, -0.0428597666, -0.0658241659, -0.114456557, -0.106830753, -0.0586995706, 0.0279622488, 0.0323923454, -0.00418315269, -0.131964132, -0.0308927745, -0.0672691539, 0.0376390964, -0.0317809209, -0.147463486, -0.0706574917, 0.0185221247, 0.132252961, -0.158320606, 0.026732469, -0.10199368, -0.0534288362, -0.0309845041, 0.100389093, -0.134254992, 0.00933926925, -0.046615012, -0.12006966, 0.0782608092, 0.0736895055, 0.0822508186, -0.0227471944, 0.0878217146, -0.137264773, -0.1176171, 0.0138121042, 0.0491721779, 0.0136306696, -0.090548791, 0.0630058348, -0.136406288, -0.101197541, 0.0404558256, 0.090086326, -0.128530398, -0.226135164, 0.109265037, -0.0687788427, 0.176857248, 0.0773077458, 0.0409816019, -0.0806122348, -0.0451379567, -0.0299756341, 0.140983731, 0.00555554172, -0.0402856506, -0.084920913, -0.09508463, -0.0965267867, -0.0849358514, -0.0511886589, 0.0146661261, 0.0156131554, -0.0376326963, -0.0671210811, 0.0224287175, 0.137774587, -0.00228940486, 0.0465276316, -0.130178899, -0.149012893, 0.130293623, -0.0280530471, 0.0527597964, 0.21135141, -0.200008243, -0.0908918828, -0.0363020897, 0.0601692759, -0.0125749074, 0.0811389834, 0.17963928, 0.0170890167, 0.207968205, -0.0548401587, 0.0640945509, 0.00915475748, -0.00665144948, 0.0521441624, -0.0598076954, 0.125235885, 0.103107899, -0.0512448139, 0.0199147407, -0.102051727, 0.00533230044, 0.0623953715, -0.0797764882, -0.00129370275, 0.239951834, -0.0897608474, -0.0809930637, 0.0116302716, 0.0264315549, 0.00502448808, -0.0133893285, -0.0398890302, 0.0280222762, 0.0427577049, -0.0401622653, -0.029694058, -0.00408209302, 0.0222895369, 0.0128808133, 0.137052923, 0.00298324437, -0.0114676105, 0.0736051723, -0.140455097, 0.0202825014, -0.02705306, -0.245139763, 0.212917298, 0.104035825, 0.0293759983, -0.0546719022, -0.0314423367, -0.0398630574, -0.0343876965, 0.0905116275, -0.0775412396, -0.129571766, 0.0111265779, -0.127151802, -0.173279762, -0.0682864934, -0.0263398364, 0.0888700038, 0.209845588, 0.051952444, -0.0745497346, -0.185133874, 0.100421809, -0.0359647982, -0.100239962, 0.0507267825, 0.0249746833, -0.0182546433, 0.0273244902, -0.00399943395, -0.024655791, -0.0122731468, 0.200671896, -0.00162600097, 0.0544531643, 0.00520347059, 0.0765429288, -0.167934522, 0.111238033, 0.0929705277, -0.00967021845, -0.0453585982, -0.102070257, 0.112714708, 0.0161449425, -0.129575238, -0.0770349205, 0.0931738392, -0.0932359025, 0.115253128, -0.152637616, 0.0158179048, 0.041739326, 0.103671372, -0.0748060644, 0.0285792667, -0.011899136, -0.0192917511, 0.107791625, -0.0256559402, -0.0543608293, 0.0164244436, -0.0119684432, 0.0224394947, -0.145458579, -0.0641392097, -0.137857869, 0.0793515444, -0.0232694242, 0.0881254748, 0.139484107, 0.0756044835, 0.125058889, -0.00860834494, -0.0920527279, -0.100648604, 0.0184238963, 0.0770169795, 0.0118718268, 0.111209154, -0.113483764, 0.0125254337, -0.0266479366, -0.0571810752, 0.0200069863, 0.124276526, 0.0205191262, 0.0164585561, 0.133350834, -0.00794353709, -0.048325561, 0.0614461824, 0.0337038003, -0.113049902, 0.0363934785, -0.0499502607, 0.0158293881, 0.0611683168, 0.0159349889, -0.124337569, 0.0816555843, -0.0228196569, -0.0540381968, -0.00830301642, 0.0457908213, 0.0331352726, -0.0895112082, 0.00246492564, -0.107790858, -0.0560132973, 0.11573261, -0.0372891389, -0.111539595, -0.0485297851, -0.0968310386, -0.0706709251, 0.0666795596, -0.11741551, 0.0311872456, -0.0177999716, 0.0229795799, 0.0683093667, -0.04996939, 0.0947744995, 0.0472060777, 0.0167367272, 0.0973566622, -0.0538218617, 0.0466017947, -0.0330167077, -0.0814527273, -0.0711240023, -0.0872239992, 0.0632802621, -0.0083680097, -0.0674064085, 0.0238934588, -0.0249120407, -0.0205953475, -0.132834002, -0.155904874, -0.20259355, -0.0278226659, -0.146687314, 0.0802839473, -0.224116221, 0.0802529827, -0.0681261495, -0.0971475542, -0.00637515821, 0.0898840725, -0.0242172033, -0.0200051516, 0.0198571607, 0.0626354143, -0.0625288486, 0.0788489282, 0.0189317074, 0.185568005, 0.000117650256, -0.0706626996, -0.0232296046, 0.0265699401, -0.140608713, -0.0798913389, -0.0144935483, 0.0150925051, -0.0770403296, 0.0461982638, -0.0743894279, 0.0112759992, -0.0415325053, -0.0902260616, 0.0242120959, -0.0101395501, 0.0574476793, 0.0817934275, -0.119240142, 0.00109685957, -0.0366540477, 0.180904225, -0.0508034974, -0.0597405396, -0.00300559308, -0.0296302028, 0.0939078331, 0.0482150204, -0.00707970513, 0.0974167213, -0.0386451483, 0.0357006602, -0.0137596354, 0.202047825, -0.065607585, -0.0113760866, 0.0209448077, -0.0308414511, 0.0818564594, 0.035646081, -0.127649605, 0.105054356, 0.0557748713, 0.00202266965, -0.0665288493, 0.052466169, 0.037145067, 0.0144229438, 0.0539823025, 0.0187405162, 0.0615465529, 0.0469304807, -0.065950945, 0.0401757248, -0.0292687323, 0.158052534, 0.0467117839, -0.064893201, 0.182949245, 0.0275977291, -0.171592563, 0.06078564, -0.0222570412, 0.0590536557, -0.0516086444, 0.0321202911, -0.126681581, 0.0127856554, -0.0842492506, -0.0825054348, 0.145829186, 0.0492514409, -0.021345092, -0.0882940814, 0.219456479, -0.164974764, 0.114569366, 0.084793061, -0.0892998874, -0.0848865286, -0.0151299872, 0.10800042, -0.0836073011, -0.0394540206, -0.00415410474, 0.0545243472, 0.113440655, 0.0142033203, 0.0992297381, 0.0700212419, 0.0218305327, -0.0960413069, 0.0179279074, -0.0658347681, -0.0156512503];
    bias_0_g : ARRAY[0..31] OF REAL := [-0.581836522, 0.309231728, 0.562823296, 0.627700269, 0.377331227, 0.598591506, -0.602125108, -0.303565025, -0.210975483, -0.289409161, 0.45574379, 0.347700447, 0.275302798, -0.5403862, -0.575578272, -0.550802469, 0.286279172, -0.627842605, 0.461831361, -0.275645137, 0.570479512, -0.615097225, -0.421455711, -0.499417245, 0.348250419, 0.679803789, 0.502462208, -0.518211007, 0.372529656, 0.596038401, -0.266079992, 0.497252136];
    weights_0_o : ARRAY[0..31] OF REAL := [1.76166964, 2.15148592, 1.80391347, 1.68124664, 2.52235556, 1.41236889, 1.65919316, 1.83199465, 2.17834687, 1.65460563, 1.72433054, 2.19740796, 1.8024863, 2.31803036, 1.70240915, 1.55125129, 2.21101999, 2.17488194, 2.62146235, 2.56662989, 2.68313241, 0.862560272, 2.02623749, 1.8731904, 1.98365009, 1.40244126, 2.40513897, 1.74895322, 2.16502452, 1.9363879, 1.95291567, 2.40807748];
    recurrent_0_o : ARRAY[0..1023] OF REAL := [0.00940295961, 0.00755411293, 0.115096495, -0.042677924, -0.0687995777, -0.072212413, -0.0272679329, 0.00926187169, -0.0322404131, -0.230642751, 0.10464444, -0.118317537, 0.0643291026, -0.0847248659, -0.110454835, 0.065530844, -0.0409047455, -0.079811722, 0.0585166439, 0.0876166224, -0.0146481553, 0.0276156012, 0.0437087826, 0.0136683295, 0.122135736, -0.0417108536, 0.0472377948, -0.0826558396, -0.0739040002, -0.0169733446, -0.0704516172, -0.111660339, 0.0013261399, 0.032797996, -0.107126579, 0.051768031, 0.168218851, -0.117840573, -0.00133558537, -0.156737015, 0.00473470287, 0.0387410335, -0.0619333275, 0.0416263752, 0.158205613, 0.0598703958, 0.0712381601, -0.0656233057, 0.147444651, 0.0920717269, -0.0842068717, -0.0531333908, 0.0637576878, -0.0327701457, -0.00259020133, -6.20728533e-05, -0.0932620242, -0.136093467, -0.0542191677, -0.0130609386, -0.0714226291, -0.139094964, 0.0650555268, -0.0779461116, 0.0727291405, -0.0236136429, 0.0512026139, -0.101979688, 0.00239524571, 0.0366442576, -0.0302348658, 0.0942990929, -0.0132932235, -0.0642298311, 0.0192060657, 0.0130893327, 0.101625614, 0.200168759, 0.0517889932, -0.108799636, 0.104390532, -0.0586065203, -0.163236856, 0.0647632331, -0.0528851151, -0.107174575, 0.0846626312, 0.037532419, -0.049235642, -0.0950798392, 0.191777244, 0.0884989724, 0.000524577685, -0.0158200487, -0.0106198462, -0.102214061, 0.0069015082, -0.0446161591, -0.0392294414, 0.0153008103, -0.027325429, -0.0261812173, 0.0347592905, -0.0386674777, -0.0300151668, 0.002856954, -0.00180103246, 0.0520746112, -0.00637343619, -0.028616976, 0.0337644443, -0.0843739882, 0.0802535638, -0.0490648001, -0.0998648554, 0.0383425839, -0.0290285107, 0.145915732, 0.00134465739, 0.101120107, 0.182724848, 0.138152152, 0.0405496918, -0.0204477198, 0.0529464185, 0.049938079, 0.0684493631, 0.065276593, -0.00253880629, -0.0155425929, -0.037788067, -0.0378959365, 0.0827185288, -0.164564133, 0.0313715376, 0.0749724954, -0.0116761904, 0.0597785451, 0.0476476401, 0.108241357, -0.0507849157, -0.077297315, -0.00137838325, 0.059471447, 0.0385285877, -0.0541518517, 0.0803878233, 0.0667919442, -0.0593200326, -0.0991778895, 0.0175430924, 0.0742868111, 0.0518188477, 0.00270438683, 0.00619300222, -0.0744272992, 0.04556676, -0.0101611707, -0.0633157417, 0.0911582336, 0.0333724804, 0.0274891406, 0.090359278, -0.0250894763, -0.0330442227, 0.0266552437, 0.119048312, 0.0323781371, -0.0843255669, 0.136369541, -0.0256569721, -0.0414893776, 0.0121494886, -0.00654248102, 0.0232459698, -0.00572938658, -0.0533263944, -0.226630121, -0.157875374, 0.0423009694, -0.0904081017, -0.0658113956, -0.151652411, 0.0201764442, -0.0914419144, -0.221003428, -0.00242811069, -0.0150172506, 0.00472717499, 0.025153067, 0.0449665263, -0.00235806056, 0.079561159, -0.00979024544, -0.032114543, -0.0120351668, -0.0658440515, -0.0523885936, 0.0321432129, -0.0523841158, 0.0984722227, -0.0391403213, -0.144826144, -0.0854723975, 0.00218068436, -0.0135808857, -0.03519921, -0.000386994798, -0.0123389661, -0.0385522321, -0.0213163309, 0.0617649332, 0.0749436319, 0.0909294337, 0.0126738595, -0.0654598102, -0.0385108218, -0.0317040943, -0.109090902, 0.0275919586, -0.0637576133, 0.0479899794, -0.0208571032, 0.0530534722, -0.0127447946, 0.0714634806, 0.0186050329, 0.132866919, 0.047393024, -0.164494514, -0.0709982663, -0.197920769, -0.0988798514, -0.154706299, -0.00919868704, 0.135501906, -0.0794674754, 0.0428844541, -0.0342918821, -0.00617858162, 0.0376018286, -0.0680695921, 0.0221220106, 0.0718257576, 0.118553676, -0.050622128, 0.0384315327, 0.0652998835, -0.204144284, -0.0725613013, -0.0885725841, -0.0328807719, -0.0790686682, 0.0327409133, -0.0627308935, -0.0589160621, 0.107908778, 0.105854571, 0.0165748075, -0.153165773, 0.169386417, 0.0277452115, -0.0437977612, 0.00759721361, -0.0423627906, 0.0660784319, 0.0508499742, 0.143870711, -0.00561960228, -0.023442572, 0.0437386408, 0.00149761862, -0.000399552286, -0.0776806548, -0.0184591748, -0.0243691169, 0.0632502511, 0.0728501529, 0.22410582, -0.0715147927, 0.0263980404, 0.0661763474, 0.0158529393, -0.104689792, 0.141211525, -0.115490779, -0.104434364, -0.0153036872, 0.0917724967, 0.0325791463, -0.0241213962, 0.102279559, 0.0870001167, 0.168846309, -0.0263923127, -0.0943953693, -0.0341686681, -0.103419013, -0.0506225117, 0.0443563312, 0.0734882578, -0.20514065, 0.0447646864, 0.165888399, -0.128757671, -0.0927457958, 0.0178062543, -0.162450165, -0.0262432843, 0.0825252756, -0.0787173957, -0.040292982, -0.108019806, -0.0473746732, -0.0170018319, -0.0375407748, 0.020163184, -0.16951406, -0.0577934161, 0.121143833, -0.166133866, 0.00333427079, -0.0296162926, 0.0398686938, 0.0665326789, 0.00922309794, -0.0551782735, 0.0244766846, -0.0628519878, -0.04631681, -0.0722112879, 0.0116234832, -0.0296955295, 0.0324297883, -0.130168721, 0.0592515282, 0.116192907, -0.0726454109, -0.0396480337, 0.0916632488, -0.104579613, -0.0471825674, -0.122244224, 0.081308797, 0.193325117, 0.189926103, -0.0254899431, 0.0820645839, 0.0491590649, -0.136623114, 0.0501643419, 0.0898105651, 0.00516937859, 0.0155608766, -0.0546327084, 0.0111690732, -0.0464842953, -0.00988538377, 0.0777462199, -0.092872113, 0.00941140018, -0.0898972526, 0.0452392437, -0.0379958972, -0.0256155878, 0.00121246767, 0.122499265, -0.155646548, 0.137311667, 0.0531266965, -0.0224689916, -0.148353025, 0.0808101892, 0.000106146748, -0.0536474399, 0.113646872, -0.0760857239, 0.100148708, 0.104765221, -0.127270341, 0.119741932, 0.0984719768, -0.0625462756, 0.0391485877, -0.0977053046, 0.0311810058, 0.122336999, 0.0991463363, -0.152850673, -0.126814917, 0.137886658, 0.0196889862, 0.00036867708, -0.041853752, 0.00032799691, -0.0285460465, 0.0504141301, 0.0104170991, -0.088729918, 0.148330212, -0.132904887, -0.193576798, -0.0709711909, -0.0887464732, -0.0169851165, -0.173731774, 0.0608291142, -0.0309687927, 0.0319064818, 0.00807518139, -0.0315297581, -0.0107264407, 0.0538853444, -0.0256053619, 0.0379964188, 0.114215061, 0.102790691, 0.0162327755, -0.0697668716, -0.0459094904, 0.041000735, -0.0303599257, 0.0214464925, 0.0471011922, -0.0483245775, -0.0823166221, 0.115071237, -0.0598229952, -0.136108965, -0.0884952694, -0.0799057409, -0.0798797309, -0.0112735564, 0.136234418, 0.00894561596, 0.0112956567, -0.146669015, -0.0146678369, -0.0345497392, 0.0654982701, 0.139236867, 0.0877570882, 0.00425055996, -0.0335871018, -0.055470705, -0.119062744, -0.0217707735, -0.0317912698, -0.0557364263, 0.0064813341, 0.0346823484, 0.0402181335, -0.0795349181, -0.0339652523, -0.0621741228, -0.0346614681, -0.0791338608, -0.0203673076, 0.0533535257, -0.0210802741, 0.0295632184, 0.122478977, 0.0386940502, 0.0747209564, -0.035176415, -0.0267058909, 0.0508651286, 0.124386981, 0.00834561139, -0.0229657106, -0.0362279378, -0.0746846721, 0.1526604, -0.0690576956, 0.0766654983, -0.0125717577, -0.00264364225, -0.0555995144, -0.0714724436, 0.0160994511, -0.0711663812, 0.0451494791, -0.0155628053, 0.0778531507, 0.0541700236, -0.0627987236, -0.0475395247, 0.0483013168, 0.130044609, 0.00148523226, -0.000589112751, -0.216675207, 0.0445254482, 0.0251138806, 0.186854556, 0.0237812288, 0.0635370985, -0.0794747323, 0.00265040062, -0.0580378696, -0.0826012269, 0.00483027613, 0.0144991651, 0.0774491727, 0.103358947, -0.0419588909, -0.0418315418, 0.00249775359, 0.0570190549, 0.0287894029, -0.196899518, -0.0413676202, 0.0729663298, 0.111533113, -0.0416263677, -0.0190843474, 0.00833295658, 0.0728022307, -0.0798861906, -0.142964661, 0.189616278, 0.107266553, 0.0479326174, -0.0513671115, 0.0100198779, -0.0526829064, 0.0140956752, 0.133747742, -0.100496694, -0.0458974093, -0.17136392, 0.0560829677, 0.124964803, 0.0985248983, 0.147003263, -0.046480041, 0.0214077495, -0.0132091092, 0.0207870677, 0.0835642815, 0.0817925781, -0.170143887, 0.17362538, 0.0743283778, -0.0321706645, 0.0925798416, 0.0761633515, 0.00363507261, 0.00698193442, 0.0864529088, 0.0134779243, 0.130662471, 0.0188912973, -0.0890371948, 0.0135746505, -0.0819012225, -0.0561677404, 0.0858705565, 0.134336963, 0.0731528774, 0.0668139905, -0.00727270171, -0.171155855, -0.176729947, 0.157706946, -0.00370704569, -0.019415535, 0.0139584728, -0.0511804596, 0.0156400725, -0.0629388541, 0.112680107, 0.0523111597, 0.0331060924, 0.00067013409, 0.0274387877, -0.0903706104, -0.137830764, -0.074579224, -0.0242071804, 0.115067095, -0.203831613, 0.0286178365, -0.10884963, 0.0916968584, 0.0467169657, -0.0504168309, -0.00738107692, 0.084313944, 0.00739513617, -0.138974085, -0.0421721563, -0.105397157, -0.0408358052, -0.0923688188, 0.149557367, -0.0459497124, 0.0647480488, -0.0152704371, -0.0507107601, 0.0107343039, 0.0556540638, 0.00192478346, -0.0172670968, 0.047566589, 0.0600018315, -0.166991338, -0.23060374, 0.0689732507, 0.0536555499, -0.0304665528, 0.0756664574, 0.0230779555, -0.0165151916, -0.0299490094, 0.205423892, 0.0773955211, -0.0700185001, -0.092860885, 0.125841737, 0.0942816362, -0.000334034296, 0.0888635069, 0.134790957, 0.00952864066, -0.0130817145, -0.0113518434, 0.0765872896, -0.046991799, 0.0565642603, -0.10095264, 0.0415524058, 0.0689811036, -0.161537424, -0.0776354969, 0.00139015773, 0.0846884474, -0.00426580478, 0.0122183012, -0.137453079, 0.0109542022, 0.0643141791, -0.0345648713, -0.0716342479, -0.0267292559, 0.0528225079, -0.0488730147, -0.0978596509, 0.0690070018, 0.0377497748, 0.260566741, -0.0211947244, 0.0902764276, -0.0760704279, -0.165018231, 0.0914126858, -0.109231301, 0.00248528528, -0.0832909569, 0.00923062768, 0.0231752135, -0.0345980674, -0.120318428, 0.202585071, -0.0489658453, 0.0931201503, 0.00296919793, 0.00408220943, -0.0654315427, 0.0775531456, -0.0809141994, -0.163404346, -0.0341040231, -0.00910625234, -0.0850221962, 0.0496852919, -0.00401834678, -0.00325406063, -0.0136100044, -0.111735515, 0.138105169, 0.00394274434, -0.0974463373, -0.0238440223, 0.0086933719, 0.0330760479, 0.0655094534, -0.0967422575, 0.0312708318, 0.0540803261, 0.00790893938, 0.0864191577, -0.0839207917, 0.0384440944, -0.00443800678, 0.137406886, 0.151308134, 0.00196464593, -0.0475457311, 0.0574964359, -0.0727273971, -0.0649731159, -0.185732558, 0.0244781822, -0.0571265817, -0.0532686077, -0.0147761256, 0.0467458963, 0.0950350761, 0.0823343769, -0.159491122, 0.158860147, 0.146393508, 0.108601041, 0.00771425664, 0.0991985947, 0.0832471102, -0.103699535, 0.076454632, -0.16798152, -0.0433627702, -0.0173479766, 0.0667291805, 0.0684928745, -0.130805522, 0.13434194, 0.187706485, -0.00418429356, -0.0683465153, 0.0159462877, 0.190812469, 0.00438944763, 0.059258882, -0.0358963646, -0.0699237064, 0.0436176211, 0.066850923, -0.0999275967, -0.018887518, 0.0987434164, -0.109033436, 0.0815993696, 0.0886577591, 0.0298503656, -0.0935864151, -0.0950844064, -0.0403584018, 0.00264140614, -0.0686242282, -0.0333514996, -0.100879706, 0.0649337992, -0.0236066375, 0.0720798448, -0.129186526, -0.0869132876, -0.0932245404, 0.0376013368, 0.0628137365, -0.0166926272, 0.0620947145, 0.0991740674, -0.112504482, 0.0483920723, 0.0436216854, 0.0281163547, -0.0870263651, -0.00127254054, 0.0989212766, 0.00918210484, 0.0137481522, 0.264207333, -0.111050501, -0.0150859188, -0.0475890525, 0.0811483115, 9.45646316e-05, -0.00627101492, -0.054559771, 0.0186051261, -0.00254060701, -0.0535421669, -0.0268133804, -0.0900333375, -0.103259884, 0.0176316574, 0.130949154, -0.0384676009, 0.100820087, 0.0735955909, -0.0995612741, -0.0913044661, -0.121986471, 0.0186118782, -0.0619993471, -0.0487035885, 0.0575196259, -0.0171687901, -0.0586452633, -0.210880727, -0.0571339205, -0.0890654996, -0.057956472, -0.0960246027, 0.043735899, 0.121598385, 0.0576094538, 0.0753752664, -0.0079896776, -0.0422117412, -0.0296790861, -0.0247896053, 0.0732908472, 0.163666651, -0.102933981, 0.122965246, 0.00858018361, -0.0385209695, -0.00498644449, -0.00461675785, 0.0330602862, 0.064378418, 0.0656299144, -0.00960236229, -0.0972309783, -0.108714014, 0.000549951103, 0.0859012976, 0.0260656364, -0.034032993, -0.0195725467, 0.0440910757, 0.12195576, 0.0417411812, 0.0281464849, -0.00667279027, 0.062305741, 0.0481587239, -0.0517128482, 0.17757614, 0.0856081247, -0.130525604, 0.103785418, 0.055400975, 0.0732730702, 0.0942987725, 0.0392186344, 0.0967030972, 0.175165057, 0.12192104, 0.112133734, 0.0404777713, 0.00404247548, -0.0719789937, -0.13364166, -0.0715420321, -0.112084597, -0.0762356967, 0.181123614, -0.109189495, 0.0228723157, -0.0230852216, 0.0559163019, 0.019585643, -0.0351398773, 0.111536123, -0.00649681594, -0.0334636979, -0.0826677606, -0.0509850308, 0.0268876087, -0.0169348698, -0.0222709831, -0.0280623194, 0.186100706, 0.116426975, -0.0163961202, -0.0839308649, -0.138978466, -0.100841418, 0.12822099, 0.163865507, -0.0214711688, 0.132302761, -0.0400597639, -0.0819613189, -0.0610583723, 0.0967052653, 0.078920044, -0.0981773213, -0.080126062, -0.0581553467, 0.19589673, -0.129951239, -0.148484752, 0.0907548368, -0.197615057, -0.0573443063, 0.0216115937, 0.195829257, 0.143931389, 0.0198122784, 0.0769877732, 0.0376244411, 0.0296427533, 0.16869539, 0.238671884, 0.0231687501, -0.00167449564, -0.0890486091, -0.146714061, -0.0778311715, -0.0524697006, -0.023846712, 0.0714461803, 0.11033161, -0.0360278338, -0.0077593727, 0.075854592, 0.0122237653, -0.00860917568, -0.0719976574, -0.0513389856, -0.0889469236, -0.105406053, -0.00969936885, 0.0439453907, 0.146225467, 0.0669558123, -0.0317291021, -0.0612652041, -0.0401737615, 0.00219145953, 0.0208743997, -0.0458788611, -0.0464125834, 0.00208988134, -0.0244842246, -0.0635985881, -0.0527464822, -0.0388446599, -0.0979132652, -0.121372074, 0.154173136, -0.0304308217, 0.0579602383, -0.0668197349, -0.110516854, -0.0324362293, 0.0505200103, -0.0427619889, 0.0436151326, 0.0123298597, -0.0453848541, 0.0577095225, 0.00519362558, 0.01615992, -0.0817289129, 0.142530143, -0.195396483, -0.0857854933, -0.123143569, 0.0672932565, 0.192832798, -0.00114903413, 0.0115235765, -0.0716098472, -0.0871109217, 0.123212636, 0.0870620012, -0.0497699864, -0.0373518653, -0.022611212, 0.127774164, -0.132909119, -0.0457881801, -0.0781681389, 0.0702276602, -0.018564729, 0.031530641, -0.000962574501, -0.228418514, 0.153743595, -0.0932296216, -0.0485839546, -0.0550276376, 0.0493867695, -0.0254413243, 0.0940306783, -0.0330990031, 0.0261724368, -0.0490734018, 0.0402796119, 0.0260037147, -0.220740169, -0.0712086633, 0.103645191, 0.0819230452, -0.00590606639, -0.0805149823, -0.026218554, 0.0562471673, -0.163178831, -0.0579855554, -0.00015405193, -0.0783496872, -0.158449441, 0.0623654053, 0.0785555393, 0.103969418, -0.127964616, 0.0210935604, -0.216164395, -0.12698108, -0.00314846588, -0.188199058, 0.0155188572, -0.0197393261, -0.0456314236, 0.0123809148, 0.0702180862, -0.0450024381, -0.0358816199, 0.0312396828];
    bias_0_o : ARRAY[0..31] OF REAL := [2.29764819, 2.28623676, 2.31636786, 2.33543444, 2.41648626, 2.18064857, 2.36472201, 2.09292531, 1.96772707, 1.97798216, 2.35417676, 2.41789675, 2.00718355, 2.6219213, 2.27783322, 2.34042072, 2.58982182, 2.62811208, 2.81970739, 2.30013108, 2.70701814, 2.25743461, 2.46817327, 2.4693501, 2.27841878, 2.32868433, 2.73383212, 2.39126229, 2.39541388, 2.6857779, 2.02658653, 2.60208464];

    weights_4 : ARRAY[0..95] OF REAL := [-1.94196701, -0.620840371, 2.74082971, 2.6686244, -0.920595706, -1.77902639, 2.17973971, 0.663026094, -2.88496447, 1.65780127, 0.738997638, -2.63572311, 3.19554853, -0.842667878, -2.54104638, 1.83732128, 0.613951564, -2.50140095, -2.02277255, -0.920283854, 2.55350661, -2.42575645, 0.992404461, 1.56410694, -2.42463088, 1.1175524, 1.59520495, -2.41728258, 0.856007397, 1.49977267, 2.5576663, -0.118251927, -2.93316603, 2.97396612, -0.759401917, -1.67675328, 2.08135438, -1.07170939, -1.49270475, -2.41047621, -0.156935126, 3.04320097, -2.00978017, -0.665324509, 2.68710613, -2.18492866, -0.476125509, 2.77966881, 3.01413131, -1.1779381, -2.24001884, -1.87072659, -0.826954484, 2.8566947, 2.6916151, -0.979066253, -2.69893408, -2.56666899, 1.02631879, 1.68065679, 2.95961666, -0.0735915527, -2.38677359, -1.01507854, -0.342460603, 1.9419167, -2.69065309, 0.872575521, 2.30487227, -2.41596532, 0.415328234, 2.07724428, 2.39219975, -0.887224913, -1.97632694, 1.60756791, 0.677681327, -2.30569506, 2.71840882, -0.804784656, -2.71014643, -2.58443522, -0.320526242, 2.39582062, 2.80470943, -0.523335159, -1.50438273, 1.69906557, 0.587613523, -3.0326252, -2.54614258, 0.895354331, 1.99043202, 2.9209516, -0.233491495, -2.13559628];
    bias_4 : ARRAY[0..2] OF REAL := [0.0396483429, 0.343401939, -0.643289447];

END_VAR

VAR
    (* Merged variables from all regions *)
    buffer_0 : ARRAY[0..31] OF REAL;
    buffer_1 : ARRAY[0..31] OF REAL;
    c_state_0 : ARRAY[0..31] OF REAL;
    f_gate_0 : ARRAY[0..31] OF REAL;
    g_gate_0 : ARRAY[0..31] OF REAL;
    h_state_0 : ARRAY[0..31] OF REAL;
    i_gate_0 : ARRAY[0..31] OF REAL;
    o_gate_0 : ARRAY[0..31] OF REAL;

    (* Temporary computation variables *)
    i : DINT;
    j : DINT;
    t : DINT;
    sum : REAL;
    (* Computation helpers *)
    max_val : REAL;
    exp_val : REAL;
    exp_sum : REAL;
    (* Spatial loop variables *)
    oc : DINT;
    oh : DINT;
    ow : DINT;
    ic : DINT;
    kh : DINT;
    kw : DINT;
    ih : DINT;
    iw : DINT;
END_VAR

(* Forward pass execution *)

(* Region: r0 [ACYCLIC] *)
(* Acyclic Region r0 *)
(* Layer 0: LSTM (hidden_size=32, input_size=1, seq_len=1) *)
(* Generating output: Y *)

(* Initialize states to zero *)
FOR j := 0 TO 31 DO
    h_state_0[j] := 0.0;
    c_state_0[j] := 0.0;
END_FOR;

(* Process 1 timesteps *)
FOR t := 0 TO 0 DO

    (* Input Gate *)
    FOR j := 0 TO 31 DO
        sum := 0.0;
        FOR i := 0 TO 0 DO
            sum := sum + input_data * weights_0_i[j * 1 + i] ;
        END_FOR;
        FOR i := 0 TO 31 DO
            sum := sum + h_state_0[i] * recurrent_0_i[j * 32 + i] ;
        END_FOR;
    sum := sum + bias_0_i[j];
    i_gate_0[j] := 1.0 / (1.0 + EXP(-sum));
    END_FOR;

    (* Forget Gate *)
    FOR j := 0 TO 31 DO
        sum := 0.0;
        FOR i := 0 TO 0 DO
            sum := sum + input_data * weights_0_f[j * 1 + i] ;
        END_FOR;
        FOR i := 0 TO 31 DO
            sum := sum + h_state_0[i] * recurrent_0_f[j * 32 + i] ;
        END_FOR;
    sum := sum + bias_0_f[j];
    f_gate_0[j] := 1.0 / (1.0 + EXP(-sum));
    END_FOR;

    (* Cell Gate *)
    FOR j := 0 TO 31 DO
        sum := 0.0;
        FOR i := 0 TO 0 DO
            sum := sum + input_data * weights_0_g[j * 1 + i] ;
        END_FOR;
        FOR i := 0 TO 31 DO
            sum := sum + h_state_0[i] * recurrent_0_g[j * 32 + i] ;
        END_FOR;
    sum := sum + bias_0_g[j];
    exp_val := EXP(2.0 * sum);
    g_gate_0[j] := (exp_val - 1.0) / (exp_val + 1.0);
    END_FOR;

    (* Output Gate *)
    FOR j := 0 TO 31 DO
        sum := 0.0;
        FOR i := 0 TO 0 DO
            sum := sum + input_data * weights_0_o[j * 1 + i] ;
        END_FOR;
        FOR i := 0 TO 31 DO
            sum := sum + h_state_0[i] * recurrent_0_o[j * 32 + i] ;
        END_FOR;
    sum := sum + bias_0_o[j];
    o_gate_0[j] := 1.0 / (1.0 + EXP(-sum));
    END_FOR;

    (* Cell state: c_t = f_t * c_{t-1} + i_t * g_t *)
    FOR j := 0 TO 31 DO
        c_state_0[j] := f_gate_0[j] * c_state_0[j] + i_gate_0[j] * g_gate_0[j];
    END_FOR;

    (* Hidden state: h_t = o_t * tanh(c_t) *)
    FOR j := 0 TO 31 DO
        exp_val := EXP(2.0 * c_state_0[j]);
        h_state_0[j] := o_gate_0[j] * ((exp_val - 1.0) / (exp_val + 1.0));
    END_FOR;

    (* Y output: Full sequence *)
    FOR j := 0 TO 31 DO
        buffer_0[t * 32 + j] := h_state_0[j];
    END_FOR;
END_FOR;

(* Layer 1: Squeeze *)
FOR i := 0 TO 31 DO
    buffer_1[i] := buffer_0[i];
END_FOR;

(* Layer 2: Slice starts=[0] ends=[1] axes=[0] steps=[1] *)
FOR i := 0 TO 31 DO
    buffer_0[i] := buffer_1[i];
END_FOR;

(* Layer 3: Squeeze *)
FOR i := 0 TO 31 DO
    buffer_1[i] := buffer_0[i];
END_FOR;

(* Layer 4: Fused Linear + SOFTMAX *)
FOR j := 0 TO 2 DO
    sum := 0.0;
    FOR i := 0 TO 31 DO
        sum := sum + buffer_1[i] * weights_4[i * 3 + j];
    END_FOR;
output_data[j] := sum + bias_4[j];
END_FOR;

(* Softmax: find max *)
max_val := output_data[0];
FOR i := 1 TO 2 DO
    IF output_data[i] > max_val THEN
        max_val := output_data[i];
    END_IF;
END_FOR;

(* Softmax: compute exponentials and sum *)
exp_sum := 0.0;
FOR i := 0 TO 2 DO
    output_data[i] := EXP(output_data[i] - max_val);
    exp_sum := exp_sum + output_data[i];
END_FOR;

(* Softmax: normalize *)
FOR i := 0 TO 2 DO
    output_data[i] := output_data[i] / exp_sum;
END_FOR;

END_FUNCTION_BLOCK
